TYPE DUT_RECIPEPARAMETER :
STRUCT
	Value	: REAL;
END_STRUCT
END_TYPE

(* stored: Version 1.1.0.1, ProductVersion 3.1.0.25
   DUT DUT_RECIPEPARAMETER: Id {a9ae374b-2f06-44a2-9d79-a3b3880612b7} *)
